FUNCTION_BLOCK VariableToEvent (* Basic Function Block Type *)
  (* Standard: 61499-2 *)
  (* Version 0.2, 2003-12-04, JHC, Rockwell Automation, Renamed for better indexing. *)
  (* Version 0.1, 2002-11-05, JHC, Rockwell Automation, Corrected missing ST element in Algorithm REQ. *)
  (* Version 0.0, 2000-05-30, JHC, Rockwell Automation *)
  (* Compiler header: package fb.rt.cs725; *)
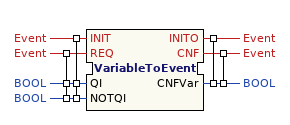
  EVENT_INPUT
    INIT WITH QI, NOTQI; (* Initialization Request *)
    REQ WITH QI, NOTQI; (* Normal Execution Request *)
  END_EVENT
  EVENT_OUTPUT
    INITO WITH CNFVar; (* Initialization Confirm *)
    CNF WITH CNFVar; (* Execution Confirmation *)
  END_EVENT
  VAR_INPUT
    QI : BOOL; (* Input event qualifier *)
    NOTQI : BOOL;
  END_VAR
  VAR_OUTPUT
    CNFVar : BOOL;
  END_VAR
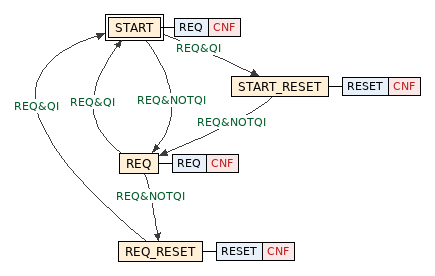
  EC_STATES
    START : REQ -> CNF; (* Initial State *)
    REQ : REQ -> CNF; (* Normal execution *)
    START_RESET : RESET -> CNF;
    REQ_RESET : RESET -> CNF;
  END_STATES
  EC_TRANSITIONS
    START TO REQ := REQ&NOTQI;
    REQ TO START := REQ&QI;
    START TO START_RESET := REQ&QI;
    REQ TO REQ_RESET := REQ&NOTQI;
    START_RESET TO REQ := REQ&NOTQI;
    REQ_RESET TO START := REQ&QI;
  END_TRANSITIONS
  ALGORITHM INIT IN Java: (* Initialization algorithm *)
CNFVar.value = true;
  END_ALGORITHM
  ALGORITHM REQ IN Java: (* Normally executed algorithm *)
CNFVar.value = true;
System.out.println(this + "                  PE CHANGED!!!");
  END_ALGORITHM
  ALGORITHM RESET IN Java:
CNFVar.value=false;
System.out.println(this+"                            PE RESET/NOT CHANGED!!!");
  END_ALGORITHM
END_FUNCTION_BLOCK
